REGION Network 4: Start Ejection
   #_w1 := #Current_machine_state = #st_finishing_molding_sub3;
   #Process_Simulation_Timers[3].TON(IN := #_w1, PT := #Process_Simulation_Timers[3].PT);
   IF #_w1 AND NOT #Process_Simulation_Timers[3].Q THEN
       "FC_change_machineState"(stop_request := #stop_request,
                               new_stateNo := #st_finishing_molding_sub3,
                               new_stateDescription := 'Mold is opening',
                               act_error_code := 0,
                               act_warning_code := 0,
                               act_stateNo => #Current_machine_state,
                               info_actStateNo => #StationInfo.StateNo,
                               info_actStateDescription => #StationInfo.StateDescription,
                               info_errorCode => #StationInfo.ErrorCode,
                               info_warningCode => #StationInfo.WarningCode);
   END_IF;
   IF #_w1 AND #Process_Simulation_Timers[3].Q THEN
       "FC_change_machineState"(stop_request := #stop_request,
                               new_stateNo := #st_cycle_completed,
                               new_stateDescription := 'Ejection is starting',
                               act_error_code := 0,
                               act_warning_code := 0,
                               act_stateNo => #Current_machine_state,
                               info_actStateNo => #StationInfo.StateNo,
                               info_actStateDescription => #StationInfo.StateDescription,
                               info_errorCode => #StationInfo.ErrorCode,
                               info_warningCode => #StationInfo.WarningCode);
   END_IF;
END_REGION
END_FUNCTION_BLOCK

// folder: Flow5_Checking_Target_Production

FUNCTION_BLOCK "FB_Checking_Target_Production"   // FB11, LAD
{ S7_Optimized_Access := 'TRUE' }
VERSION : 0.1
   VAR_INPUT
      target_quantity : UInt;
   END_VAR
   VAR_IN_OUT
      stop_request : Bool;
      Current_machine_state : UInt;
      Act_Production_Quantity : UInt;
      StationInfo : Struct
         StateNo : UInt;
         StateDescription : String;
         ErrorCode : UInt;
         ErrorDescription : String;
         WarningCode : UInt;
         WarninDescription : String;
         TotalProductionTime : Time;
         ProducedCount : UInt;
      END_STRUCT;
   END_VAR
   VAR
      temp_state : UInt;
      Timeout : Array[0..5] of IEC_TIMER;
      Process_Simulation_Timers : Array[0..20] of IEC_TIMER;
      aux_var1 : Bool;
   END_VAR
   VAR CONSTANT
      st_idle : UInt := 0;
      st_cycle_completed : UInt := 500;
      st_cycle_completed_sub1 : UInt := 501;
      st_cycle_completed_sub2 : UInt := 502;
      st_cycle_completed_sub3 : UInt := 503;
      st_cycle_completed_sub4 : UInt := 504;
      st_cycle_completed_sub5 : UInt := 505;
      st_cycle_completed_sub6 : UInt := 506;
      st_cycle_completed_sub7 : UInt := 507;
      st_cycle_completed_sub8 : UInt := 508;
      st_cycle_completed_sub9 : UInt := 509;
      st_checking_order_target : UInt := 600;
      st_checking_initial_safety : UInt := 200;
      st_order_finishing : UInt := 700;
   END_VAR
   VAR_TEMP   // added for the SCL form of the ladder/FBD networks
      _w1 : Bool;
   END_VAR
   // Process_Simulation_Timers[0].PT := T#3S;
   // Process_Simulation_Timers[1].PT := T#4S;
   // Process_Simulation_Timers[2].PT := T#10S;
   // Process_Simulation_Timers[3].PT := T#3S;
BEGIN

REGION Network 1
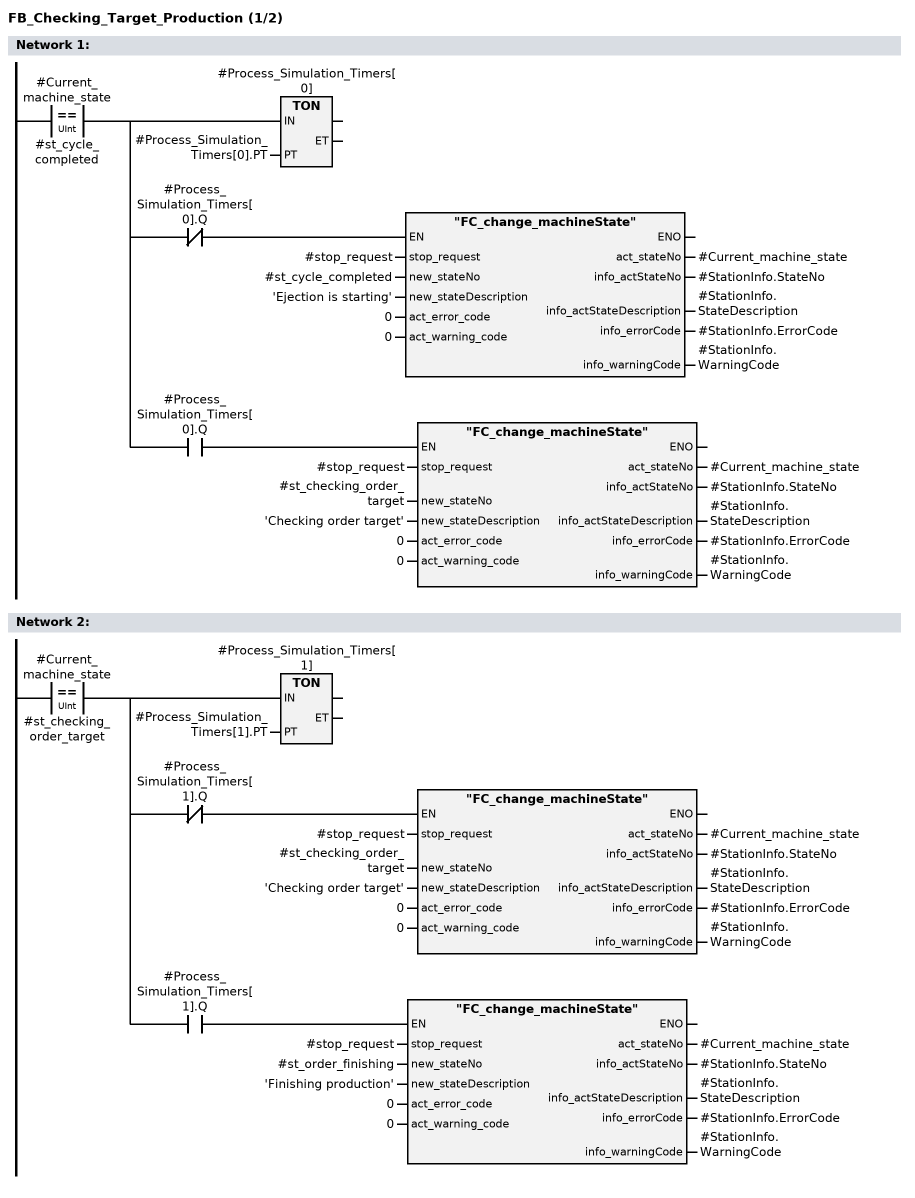
   #_w1 := #Current_machine_state = #st_cycle_completed;
   #Process_Simulation_Timers[0].TON(IN := #_w1, PT := #Process_Simulation_Timers[0].PT);
   IF #_w1 AND NOT #Process_Simulation_Timers[0].Q THEN
       "FC_change_machineState"(stop_request := #stop_request,
                               new_stateNo := #st_cycle_completed,
                               new_stateDescription := 'Ejection is starting',
                               act_error_code := 0,
                               act_warning_code := 0,
                               act_stateNo => #Current_machine_state,
                               info_actStateNo => #StationInfo.StateNo,
                               info_actStateDescription => #StationInfo.StateDescription,
                               info_errorCode => #StationInfo.ErrorCode,
                               info_warningCode => #StationInfo.WarningCode);
   END_IF;
   IF #_w1 AND #Process_Simulation_Timers[0].Q THEN
       "FC_change_machineState"(stop_request := #stop_request,
                               new_stateNo := #st_checking_order_target,
                               new_stateDescription := 'Checking order target',
                               act_error_code := 0,
                               act_warning_code := 0,
                               act_stateNo => #Current_machine_state,
                               info_actStateNo => #StationInfo.StateNo,
                               info_actStateDescription => #StationInfo.StateDescription,
                               info_errorCode => #StationInfo.ErrorCode,
                               info_warningCode => #StationInfo.WarningCode);
   END_IF;
END_REGION

REGION Network 2
   #_w1 := #Current_machine_state = #st_checking_order_target;
   #Process_Simulation_Timers[1].TON(IN := #_w1, PT := #Process_Simulation_Timers[1].PT);
   IF #_w1 AND NOT #Process_Simulation_Timers[1].Q THEN
       "FC_change_machineState"(stop_request := #stop_request,
                               new_stateNo := #st_checking_order_target,
                               new_stateDescription := 'Checking order target',
                               act_error_code := 0,
                               act_warning_code := 0,
                               act_stateNo => #Current_machine_state,
                               info_actStateNo => #StationInfo.StateNo,
                               info_actStateDescription => #StationInfo.StateDescription,
                               info_errorCode => #StationInfo.ErrorCode,
                               info_warningCode => #StationInfo.WarningCode);
   END_IF;
   IF #_w1 AND #Process_Simulation_Timers[1].Q THEN
       "FC_change_machineState"(stop_request := #stop_request,
                               new_stateNo := #st_order_finishing,
                               new_stateDescription := 'Finishing production',
                               act_error_code := 0,
                               act_warning_code := 0,
                               act_stateNo => #Current_machine_state,
                               info_actStateNo => #StationInfo.StateNo,
                               info_actStateDescription => #StationInfo.StateDescription,
                               info_errorCode => #StationInfo.ErrorCode,
                               info_warningCode => #StationInfo.WarningCode);
   END_IF;
END_REGION

REGION Network 3
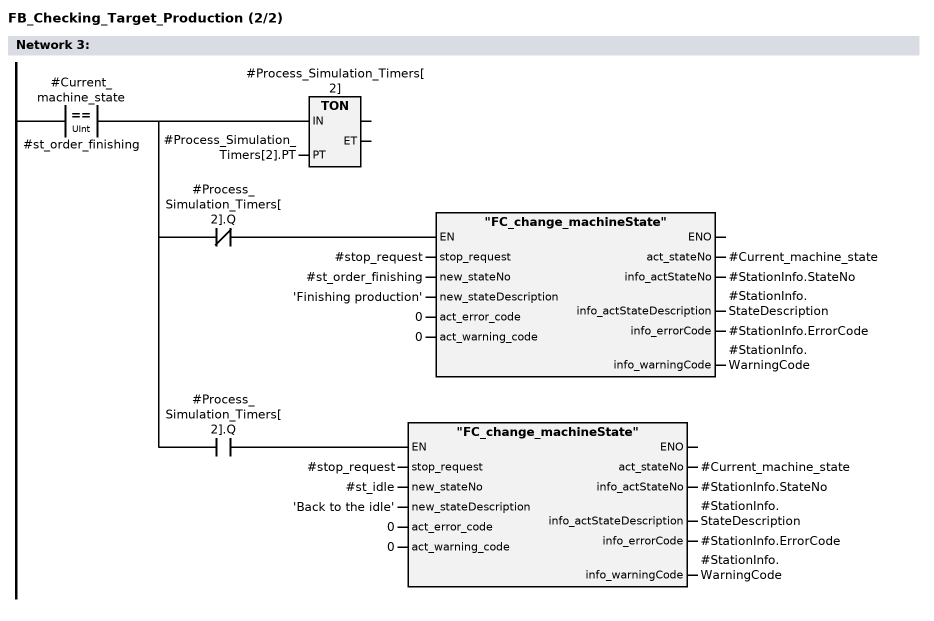
   #_w1 := #Current_machine_state = #st_order_finishing;
   #Process_Simulation_Timers[2].TON(IN := #_w1, PT := #Process_Simulation_Timers[2].PT);
   IF #_w1 AND NOT #Process_Simulation_Timers[2].Q THEN
       "FC_change_machineState"(stop_request := #stop_request,
                               new_stateNo := #st_order_finishing,
                               new_stateDescription := 'Finishing production',
                               act_error_code := 0,
                               act_warning_code := 0,
                               act_stateNo => #Current_machine_state,
                               info_actStateNo => #StationInfo.StateNo,
                               info_actStateDescription => #StationInfo.StateDescription,
                               info_errorCode => #StationInfo.ErrorCode,
                               info_warningCode => #StationInfo.WarningCode);
   END_IF;
   IF #_w1 AND #Process_Simulation_Timers[2].Q THEN
       "FC_change_machineState"(stop_request := #stop_request,
                               new_stateNo := #st_idle,
                               new_stateDescription := 'Back to the idle',
                               act_error_code := 0,
                               act_warning_code := 0,
                               act_stateNo => #Current_machine_state,
                               info_actStateNo => #StationInfo.StateNo,
                               info_actStateDescription => #StationInfo.StateDescription,
                               info_errorCode => #StationInfo.ErrorCode,
                               info_warningCode => #StationInfo.WarningCode);
   END_IF;
END_REGION
END_FUNCTION_BLOCK

// folder: Functions

FUNCTION "FC_get_time_data" : Void   // FC1, LAD
{ S7_Optimized_Access := 'TRUE' }
VERSION : 0.1
   VAR_OUTPUT
      actYear : UInt;
      actMonth : UInt;
      actDay : UInt;
      timeStamp : UDInt;
      errorGettingTime : Int;
   END_VAR
   VAR_TEMP
      timeData : DTL;
      gettingTimeState : Int;
   END_VAR
BEGIN

REGION Network 1
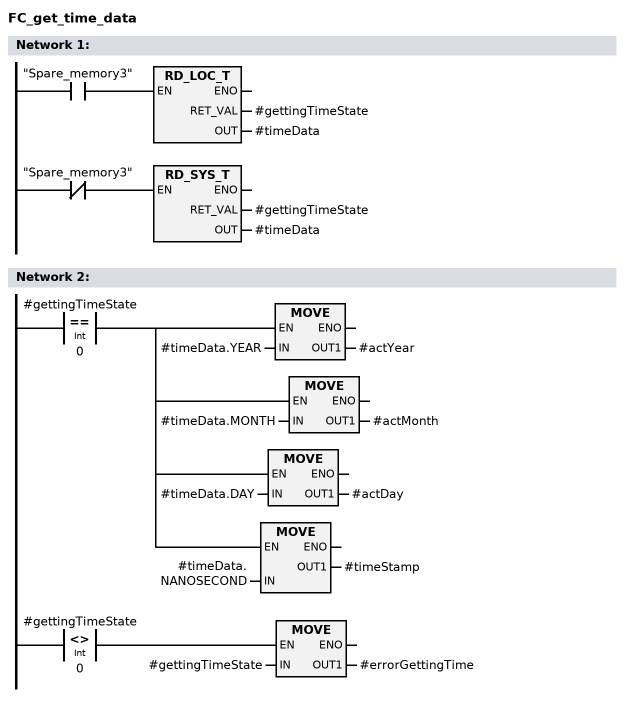
   IF "Spare_memory3" THEN #gettingTimeState := RD_LOC_T(OUT => #timeData); END_IF;
   IF NOT "Spare_memory3" THEN #gettingTimeState := RD_SYS_T(OUT => #timeData); END_IF;
END_REGION

REGION Network 2
   RUNG wire#powerrail
      { S7_Templates := "SrcType := Int" } EQ_Contact(in1 := #gettingTimeState, in2 := 0)
      wire#w1
      Move(in := #timeData.YEAR, out1 => #actYear)
   END_RUNG
   RUNG wire#w1
      Move(in := #timeData.MONTH, out1 => #actMonth)
   END_RUNG
   RUNG wire#w1
      Move(in := #timeData.DAY, out1 => #actDay)
   END_RUNG
   RUNG wire#w1
      Move(in := #timeData.NANOSECOND, out1 => #timeStamp)
   END_RUNG
   RUNG wire#powerrail
      { S7_Templates := "SrcType := Int" } NE_Contact(in1 := #gettingTimeState, in2 := 0)
      Move(in := #gettingTimeState, out1 => #errorGettingTime)
   END_RUNG
   // the same network as SCL:
   IF #gettingTimeState = 0 THEN
       #actYear := #timeData.YEAR;
       #actMonth := #timeData.MONTH;
       #actDay := #timeData.DAY;
       #timeStamp := #timeData.NANOSECOND;
   END_IF;
   IF #gettingTimeState <> 0 THEN #errorGettingTime := #gettingTimeState; END_IF;
END_REGION
END_FUNCTION

FUNCTION "FC_change_machineState" : Void   // FC2, LAD
{ S7_Optimized_Access := 'TRUE' }
VERSION : 0.1
   VAR_INPUT
      stop_request : Bool;
      new_stateNo : UInt;
      new_stateDescription : String;
      act_error_code : UInt;
      act_warning_code : UInt;
   END_VAR
   VAR_OUTPUT
      act_stateNo : UInt;
      info_actStateNo : UInt;
      info_actStateDescription : String;
      info_errorCode : UInt;
      info_warningCode : UInt;
   END_VAR
   VAR CONSTANT
      st_idle : UInt := 0;
   END_VAR
BEGIN

REGION Network 1: No Stop Request Received
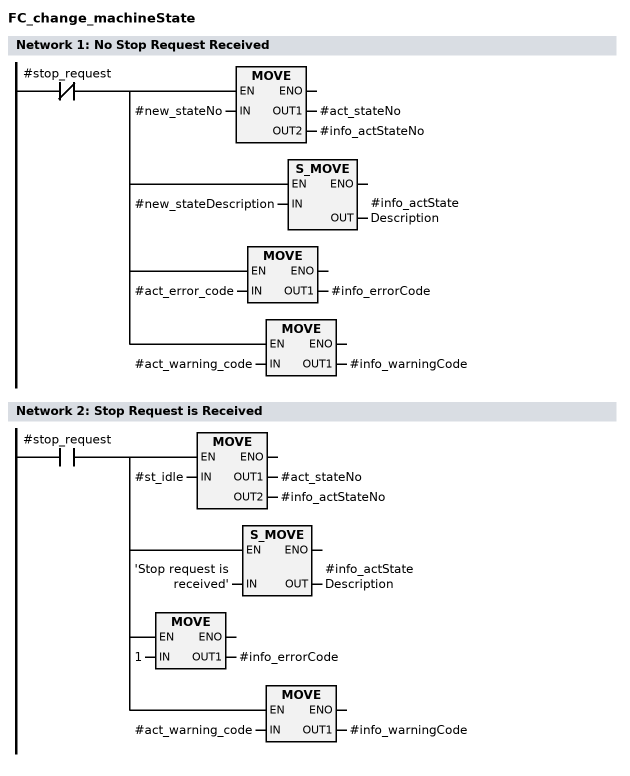
   RUNG wire#powerrail
      I_Contact( #stop_request )
      wire#w1
      Move(in := #new_stateNo, out1 => #act_stateNo, out2 => #info_actStateNo)
   END_RUNG
   RUNG wire#w1
      S_Move(in := #new_stateDescription, out => #info_actStateDescription)
   END_RUNG
   RUNG wire#w1
      Move(in := #act_error_code, out1 => #info_errorCode)
   END_RUNG
   RUNG wire#w1
      Move(in := #act_warning_code, out1 => #info_warningCode)
   END_RUNG
   // the same network as SCL:
   IF NOT #stop_request THEN
       #act_stateNo := #new_stateNo;
       #info_actStateNo := #new_stateNo;
       #info_actStateDescription := #new_stateDescription;
       #info_errorCode := #act_error_code;
       #info_warningCode := #act_warning_code;
   END_IF;
END_REGION

REGION Network 2: Stop Request is Received
   RUNG wire#powerrail
      Contact( #stop_request )
      wire#w1
      Move(in := #st_idle, out1 => #act_stateNo, out2 => #info_actStateNo)
   END_RUNG
   RUNG wire#w1
      S_Move(in := 'Stop request is received', out => #info_actStateDescription)
   END_RUNG
   RUNG wire#w1
      Move(in := 1, out1 => #info_errorCode)
   END_RUNG
   RUNG wire#w1
      Move(in := #act_warning_code, out1 => #info_warningCode)
   END_RUNG
   // the same network as SCL:
   IF #stop_request THEN
       #act_stateNo := #st_idle;
       #info_actStateNo := #st_idle;
       #info_actStateDescription := 'Stop request is received';
       #info_errorCode := 1;
       #info_warningCode := #act_warning_code;
   END_IF;
END_REGION
END_FUNCTION

// folder: Machine_transition

FUNCTION_BLOCK "FB_SubTransition"   // FB3, LAD
{ S7_Optimized_Access := 'TRUE' }
VERSION : 0.1
   VAR_INPUT
      new_state : UInt;
   END_VAR
   VAR_OUTPUT
      new_machine_state : UInt;
      previous_state_done : Bool;
   END_VAR
   VAR_IN_OUT
      stop_request : Bool;
   END_VAR
   VAR CONSTANT
      st_idle : UInt := 0;
   END_VAR
BEGIN

REGION Network 1: No Stop Request
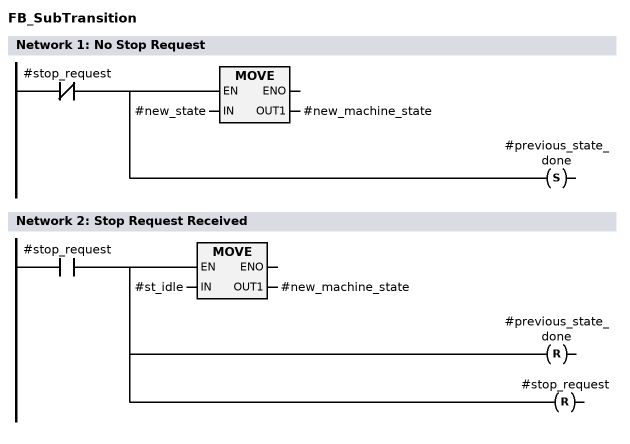
   RUNG wire#powerrail
      I_Contact( #stop_request )
      wire#w1
      Move(in := #new_state, out1 => #new_machine_state)
   END_RUNG
   RUNG wire#w1
      S_Coil( #previous_state_done )
   END_RUNG
   // the same network as SCL:
   IF NOT #stop_request THEN
       #new_machine_state := #new_state;
       #previous_state_done := TRUE;
   END_IF;
END_REGION

REGION Network 2: Stop Request Received
   RUNG wire#powerrail
      Contact( #stop_request )
      wire#w1
      Move(in := #st_idle, out1 => #new_machine_state)
   END_RUNG
   RUNG wire#w1
      R_Coil( #previous_state_done )
   END_RUNG
   RUNG wire#w1
      R_Coil( #stop_request )
   END_RUNG
   // the same network as SCL:
   IF #stop_request THEN
       #new_machine_state := #st_idle;
       #previous_state_done := FALSE;
       #stop_request := FALSE;
   END_IF;
END_REGION
END_FUNCTION_BLOCK

FUNCTION_BLOCK "FB_control_state_transition"   // FB6, LAD
TITLE = This FB sets the machine status
{ S7_Optimized_Access := 'TRUE' }
VERSION : 0.1
   VAR_INPUT
      is_start_btn_activated : Bool;
      is_stop_btn_activated : Bool;
   END_VAR
   VAR_IN_OUT
      current_machine_state : UInt;
      is_previous_state_done : Bool;
   END_VAR
   VAR
      temp_state : UInt;
      initial_temp_state : UInt;
      stop_request : Bool;
   END_VAR
   VAR CONSTANT
      st_idle : UInt := 0;
      st_checking_order : UInt := 10;
      st_checking_initial_safety : UInt := 20;
      st_checking_material_level : UInt := 30;
      st_running_molding : UInt := 40;
      st_finishing_molding : UInt := 50;
      st_cycle_completed : UInt := 60;
      st_checking_order_target : UInt := 70;
      st_order_finishing : UInt := 80;
      st_fault : UInt := 300;
   END_VAR
   VAR_TEMP   // added for the SCL form of the ladder/FBD networks
      _w1 : Bool;
   END_VAR
BEGIN

REGION Network 1: Control Stop Request
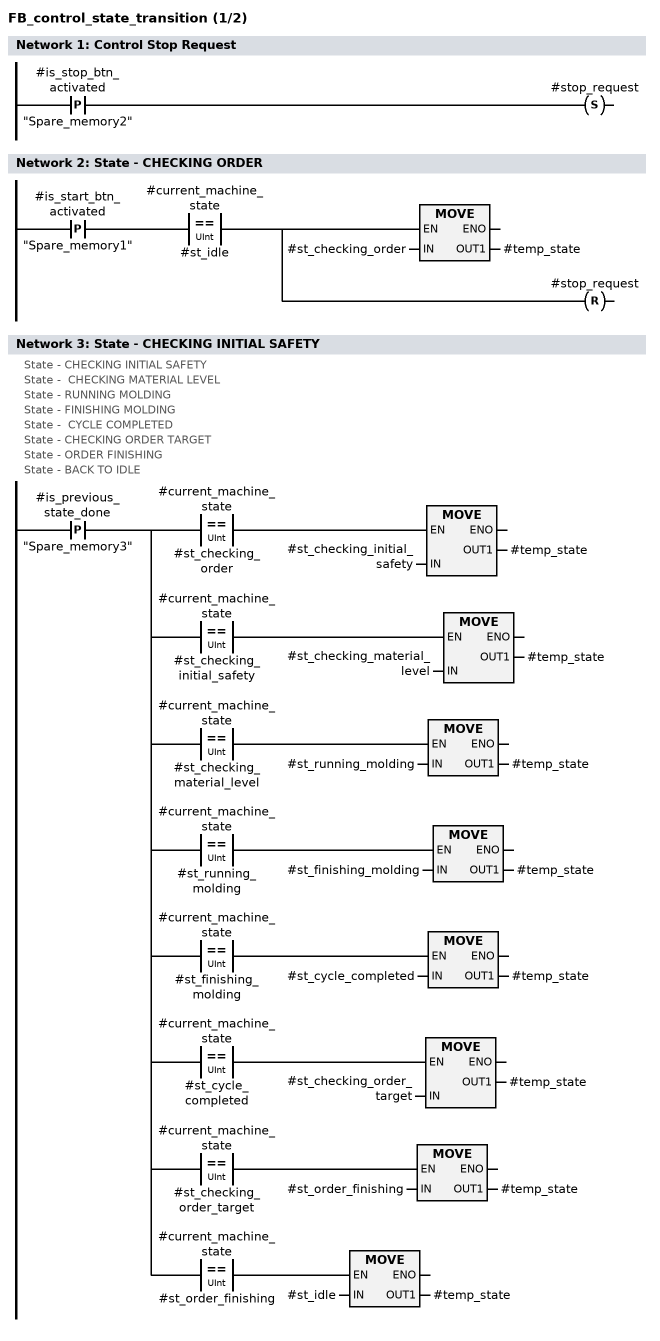
   RUNG wire#powerrail
      P_Contact(operand := #is_stop_btn_activated, bit := "Spare_memory2")
      S_Coil( #stop_request )
   END_RUNG
   // the same network as SCL:
   #_w1 := #is_stop_btn_activated AND NOT "Spare_memory2";   // rising edge of #is_stop_btn_activated
   "Spare_memory2" := #is_stop_btn_activated;
   IF #_w1 THEN #stop_request := TRUE; END_IF;
END_REGION

REGION Network 2: State - CHECKING ORDER
   RUNG wire#powerrail
      P_Contact(operand := #is_start_btn_activated, bit := "Spare_memory1")
      { S7_Templates := "SrcType := UInt" } EQ_Contact(in1 := #current_machine_state, in2 := #st_idle)
      wire#w1
      Move(in := #st_checking_order, out1 => #temp_state)
   END_RUNG
   RUNG wire#w1
      R_Coil( #stop_request )
   END_RUNG
   // the same network as SCL:
   #_w1 := #is_start_btn_activated AND NOT "Spare_memory1";   // rising edge of #is_start_btn_activated
   "Spare_memory1" := #is_start_btn_activated;
   IF #_w1 AND (#current_machine_state = #st_idle) THEN
       #temp_state := #st_checking_order;
       #stop_request := FALSE;
   END_IF;
END_REGION

REGION Network 3: State - CHECKING INITIAL SAFETY
   // State - CHECKING INITIAL SAFETY
   // State -  CHECKING MATERIAL LEVEL
   // State - RUNNING MOLDING
   // State - FINISHING MOLDING
   // State -  CYCLE COMPLETED
   // State - CHECKING ORDER TARGET
   // State - ORDER FINISHING 
   // State - BACK TO IDLE
   RUNG wire#powerrail
      P_Contact(operand := #is_previous_state_done, bit := "Spare_memory3")
      wire#w1
      { S7_Templates := "SrcType := UInt" } EQ_Contact(in1 := #current_machine_state, in2 := #st_checking_order)
      Move(in := #st_checking_initial_safety, out1 => #temp_state)
   END_RUNG
   RUNG wire#w1
      { S7_Templates := "SrcType := UInt" } EQ_Contact(in1 := #current_machine_state, in2 := #st_checking_initial_safety)
      Move(in := #st_checking_material_level, out1 => #temp_state)
   END_RUNG
   RUNG wire#w1
      { S7_Templates := "SrcType := UInt" } EQ_Contact(in1 := #current_machine_state, in2 := #st_checking_material_level)
      Move(in := #st_running_molding, out1 => #temp_state)
   END_RUNG
   RUNG wire#w1
      { S7_Templates := "SrcType := UInt" } EQ_Contact(in1 := #current_machine_state, in2 := #st_running_molding)
      Move(in := #st_finishing_molding, out1 => #temp_state)
   END_RUNG
   RUNG wire#w1
      { S7_Templates := "SrcType := UInt" } EQ_Contact(in1 := #current_machine_state, in2 := #st_finishing_molding)
      Move(in := #st_cycle_completed, out1 => #temp_state)
   END_RUNG
   RUNG wire#w1
      { S7_Templates := "SrcType := UInt" } EQ_Contact(in1 := #current_machine_state, in2 := #st_cycle_completed)
      Move(in := #st_checking_order_target, out1 => #temp_state)
   END_RUNG
   RUNG wire#w1
      { S7_Templates := "SrcType := UInt" } EQ_Contact(in1 := #current_machine_state, in2 := #st_checking_order_target)
      Move(in := #st_order_finishing, out1 => #temp_state)
   END_RUNG
   RUNG wire#w1
      { S7_Templates := "SrcType := UInt" } EQ_Contact(in1 := #current_machine_state, in2 := #st_order_finishing)
      Move(in := #st_idle, out1 => #temp_state)
   END_RUNG
   // the same network as SCL:
   #_w1 := #is_previous_state_done AND NOT "Spare_memory3";   // rising edge of #is_previous_state_done
   "Spare_memory3" := #is_previous_state_done;
   IF #_w1 AND (#current_machine_state = #st_checking_order) THEN
       #temp_state := #st_checking_initial_safety;
   END_IF;
   IF #_w1 AND (#current_machine_state = #st_checking_initial_safety) THEN
       #temp_state := #st_checking_material_level;
   END_IF;
   IF #_w1 AND (#current_machine_state = #st_checking_material_level) THEN
       #temp_state := #st_running_molding;
   END_IF;
   IF #_w1 AND (#current_machine_state = #st_running_molding) THEN
       #temp_state := #st_finishing_molding;
   END_IF;
   IF #_w1 AND (#current_machine_state = #st_finishing_molding) THEN
       #temp_state := #st_cycle_completed;
   END_IF;
   IF #_w1 AND (#current_machine_state = #st_cycle_completed) THEN
       #temp_state := #st_checking_order_target;
   END_IF;
   IF #_w1 AND (#current_machine_state = #st_checking_order_target) THEN
       #temp_state := #st_order_finishing;
   END_IF;
   IF #_w1 AND (#current_machine_state = #st_order_finishing) THEN #temp_state := #st_idle; END_IF;
END_REGION

REGION Network 4: Set the current machine state to new state value
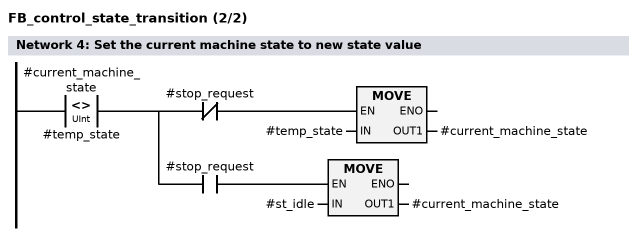
   RUNG wire#powerrail
      { S7_Templates := "SrcType := UInt" } NE_Contact(in1 := #current_machine_state, in2 := #temp_state)
      wire#w1
      I_Contact( #stop_request )
      Move(in := #temp_state, out1 => #current_machine_state)
   END_RUNG
   RUNG wire#w1
      Contact( #stop_request )
      Move(in := #st_idle, out1 => #current_machine_state)
   END_RUNG
   // the same network as SCL:
   #_w1 := #current_machine_state <> #temp_state;
   IF #_w1 AND NOT #stop_request THEN #current_machine_state := #temp_state; END_IF;
   IF #_w1 AND #stop_request THEN #current_machine_state := #st_idle; END_IF;
END_REGION
END_FUNCTION_BLOCK

// folder: Manage_outputs

FUNCTION_BLOCK "FB_manage_outputs"   // FB8, LAD
{ S7_Optimized_Access := 'TRUE' }
VERSION : 0.1
BEGIN

REGION Network 1: Feeder_Start
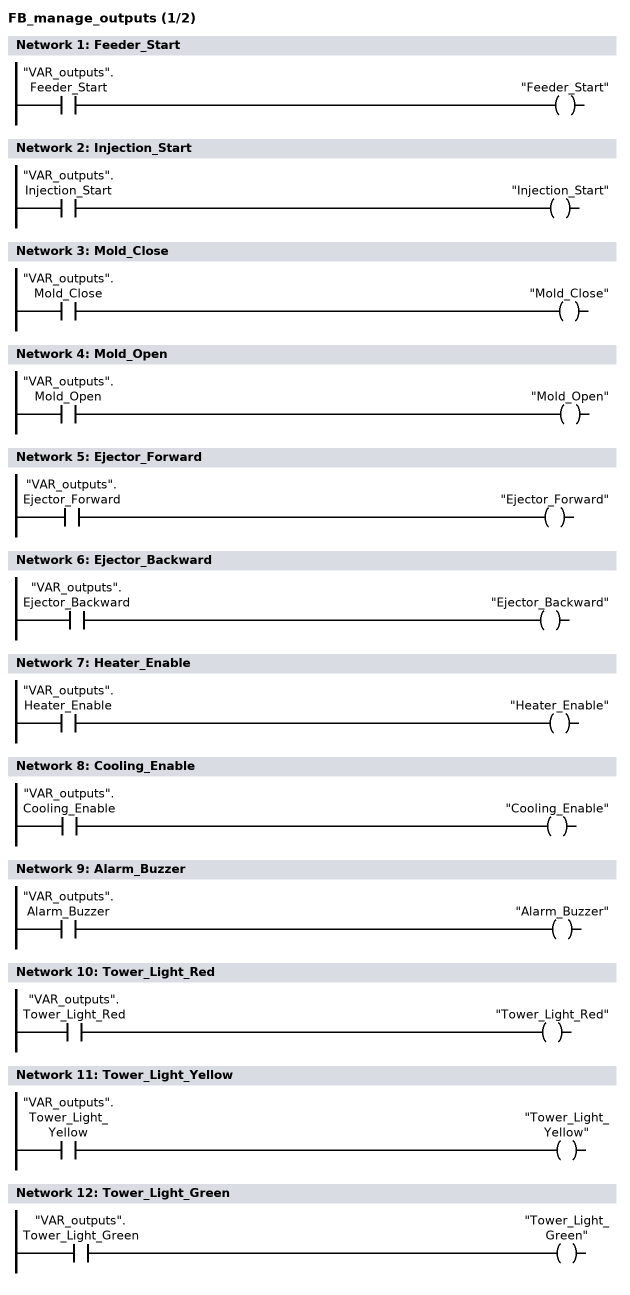
   RUNG wire#powerrail
      Contact( "VAR_outputs".Feeder_Start )
      Coil( "Feeder_Start" )
   END_RUNG
   // the same network as SCL:
   "Feeder_Start" := "VAR_outputs".Feeder_Start;
END_REGION

REGION Network 2: Injection_Start
   RUNG wire#powerrail
      Contact( "VAR_outputs".Injection_Start )
      Coil( "Injection_Start" )
   END_RUNG
   // the same network as SCL:
   "Injection_Start" := "VAR_outputs".Injection_Start;
END_REGION

REGION Network 3: Mold_Close
   RUNG wire#powerrail
      Contact( "VAR_outputs".Mold_Close )
      Coil( "Mold_Close" )
   END_RUNG
   // the same network as SCL:
   "Mold_Close" := "VAR_outputs".Mold_Close;
END_REGION

REGION Network 4: Mold_Open
   RUNG wire#powerrail
      Contact( "VAR_outputs".Mold_Open )
      Coil( "Mold_Open" )
   END_RUNG
   // the same network as SCL:
   "Mold_Open" := "VAR_outputs".Mold_Open;
END_REGION

REGION Network 5: Ejector_Forward
   RUNG wire#powerrail
      Contact( "VAR_outputs".Ejector_Forward )
      Coil( "Ejector_Forward" )
   END_RUNG
   // the same network as SCL:
   "Ejector_Forward" := "VAR_outputs".Ejector_Forward;
END_REGION

REGION Network 6: Ejector_Backward
   RUNG wire#powerrail
      Contact( "VAR_outputs".Ejector_Backward )
      Coil( "Ejector_Backward" )
   END_RUNG
   // the same network as SCL:
   "Ejector_Backward" := "VAR_outputs".Ejector_Backward;
END_REGION

REGION Network 7: Heater_Enable
   RUNG wire#powerrail
      Contact( "VAR_outputs".Heater_Enable )
      Coil( "Heater_Enable" )
   END_RUNG
   // the same network as SCL:
   "Heater_Enable" := "VAR_outputs".Heater_Enable;
END_REGION

REGION Network 8: Cooling_Enable
   RUNG wire#powerrail
      Contact( "VAR_outputs".Cooling_Enable )
      Coil( "Cooling_Enable" )
   END_RUNG
   // the same network as SCL:
   "Cooling_Enable" := "VAR_outputs".Cooling_Enable;
END_REGION

REGION Network 9: Alarm_Buzzer
   RUNG wire#powerrail
      Contact( "VAR_outputs".Alarm_Buzzer )
      Coil( "Alarm_Buzzer" )
   END_RUNG
   // the same network as SCL:
   "Alarm_Buzzer" := "VAR_outputs".Alarm_Buzzer;
END_REGION

REGION Network 10: Tower_Light_Red
   RUNG wire#powerrail
      Contact( "VAR_outputs".Tower_Light_Red )
      Coil( "Tower_Light_Red" )
   END_RUNG
   // the same network as SCL:
   "Tower_Light_Red" := "VAR_outputs".Tower_Light_Red;
END_REGION

REGION Network 11: Tower_Light_Yellow
   RUNG wire#powerrail
      Contact( "VAR_outputs".Tower_Light_Yellow )
      Coil( "Tower_Light_Yellow" )
   END_RUNG
   // the same network as SCL:
   "Tower_Light_Yellow" := "VAR_outputs".Tower_Light_Yellow;
END_REGION

REGION Network 12: Tower_Light_Green
   RUNG wire#powerrail
      Contact( "VAR_outputs".Tower_Light_Green )
      Coil( "Tower_Light_Green" )
   END_RUNG
   // the same network as SCL:
   "Tower_Light_Green" := "VAR_outputs".Tower_Light_Green;
END_REGION

REGION Network 13: Goto_NextStationBuffer
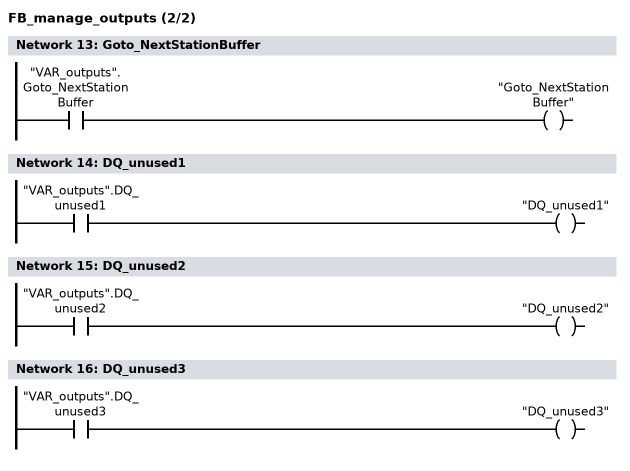
   RUNG wire#powerrail
      Contact( "VAR_outputs".Goto_NextStationBuffer )
      Coil( "Goto_NextStationBuffer" )
   END_RUNG
   // the same network as SCL:
   "Goto_NextStationBuffer" := "VAR_outputs".Goto_NextStationBuffer;
END_REGION

REGION Network 14: DQ_unused1
   RUNG wire#powerrail
      Contact( "VAR_outputs".DQ_unused1 )
      Coil( "DQ_unused1" )
   END_RUNG
   // the same network as SCL:
   "DQ_unused1" := "VAR_outputs".DQ_unused1;
END_REGION

REGION Network 15: DQ_unused2
   RUNG wire#powerrail
      Contact( "VAR_outputs".DQ_unused2 )
      Coil( "DQ_unused2" )
   END_RUNG
   // the same network as SCL:
   "DQ_unused2" := "VAR_outputs".DQ_unused2;
END_REGION

REGION Network 16: DQ_unused3
   RUNG wire#powerrail
      Contact( "VAR_outputs".DQ_unused3 )
      Coil( "DQ_unused3" )
   END_RUNG
   // the same network as SCL:
   "DQ_unused3" := "VAR_outputs".DQ_unused3;
END_REGION
END_FUNCTION_BLOCK

// folder: Simulation_data/Simulation_FB

FUNCTION_BLOCK "FB_simulate_analog_data"   // FB10, LAD
{ S7_Optimized_Access := 'TRUE' }
VERSION : 0.1
   VAR_INPUT
      Clock : Bool;
      Up : Bool;
      Down : Bool;
      TargetLevelLimit : Real;
      HighLevelLimit : Real;
      LowLevelLimit : Real;
      ResetVal : Bool;
   END_VAR
   VAR_IN_OUT
      actLevel : Real;
   END_VAR
   VAR
      value_int : Int;
      value_real : Real;
   END_VAR
   VAR_TEMP
      tag1 : Bool;
   END_VAR
   VAR CONSTANT
      incrementVal : Int := 5;
      decrementVal : Int := 150;
      normMin : Int := 0;
      normMax : Int := 27648;
   END_VAR
   VAR_TEMP   // added for the SCL form of the ladder/FBD networks
      _w1 : Bool;
   END_VAR
BEGIN

REGION Network 1: Simulate an analog input value
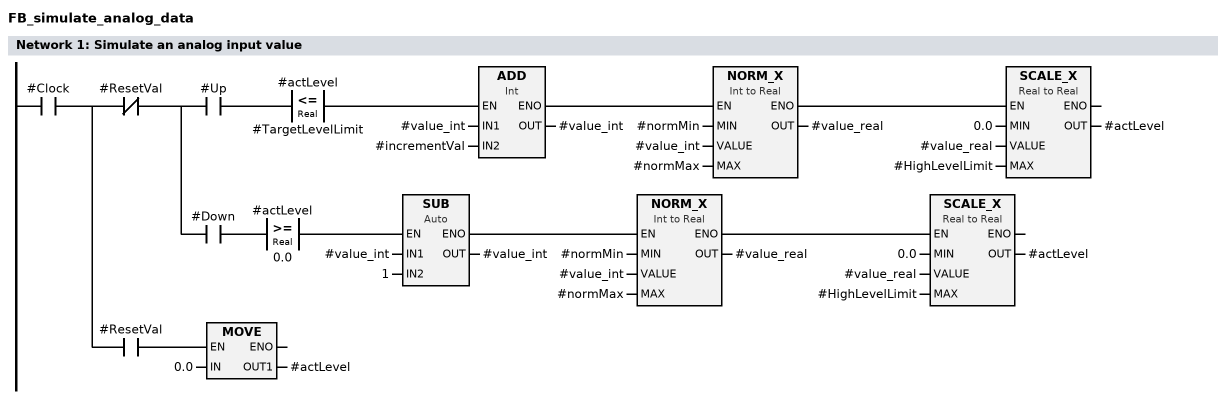
   RUNG wire#powerrail
      Contact( #Clock )
      wire#w1
      I_Contact( #ResetVal )
      wire#w2
      Contact( #Up )
      { S7_Templates := "SrcType := Real" } LE_Contact(in1 := #actLevel, in2 := #TargetLevelLimit)
      { S7_Templates := "SrcType := Int" } Add(in1 := #value_int, in2 := #incrementVal, out => #value_int)
      { S7_Templates := "[SrcType := Int, DestType := Real]" } Normalize(min := #normMin, value := #value_int, max := #normMax, out => #value_real)
      { S7_Templates := "[SrcType := Real, DestType := Real]" } Scale(min := 0.0, value := #value_real, max := #HighLevelLimit, out => #actLevel)
   END_RUNG
   RUNG wire#w2
      Contact( #Down )
      { S7_Templates := "SrcType := Real" } GE_Contact(in1 := #actLevel, in2 := 0.0)
      Sub(in1 := #value_int, in2 := 1, out => #value_int)
      { S7_Templates := "[SrcType := Int, DestType := Real]" } Normalize(min := #normMin, value := #value_int, max := #normMax, out => #value_real)
      { S7_Templates := "[SrcType := Real, DestType := Real]" } Scale(min := 0.0, value := #value_real, max := #HighLevelLimit, out => #actLevel)
   END_RUNG
   RUNG wire#w1
      Contact( #ResetVal )
      Move(in := 0.0, out1 => #actLevel)
   END_RUNG
   // the same network as SCL:
   #_w1 := #Clock AND NOT #ResetVal;
   IF #_w1 AND #Up AND (#actLevel <= #TargetLevelLimit) THEN
       #value_int := #value_int + #incrementVal;
       #value_real := NORM_X(MIN := #normMin, VALUE := #value_int, MAX := #normMax);
       #actLevel := SCALE_X(MIN := 0.0, VALUE := #value_real, MAX := #HighLevelLimit);
   END_IF;
   IF #_w1 AND #Down AND (#actLevel >= 0.0) THEN
       #value_int := #value_int - 1;
       #value_real := NORM_X(MIN := #normMin, VALUE := #value_int, MAX := #normMax);
       #actLevel := SCALE_X(MIN := 0.0, VALUE := #value_real, MAX := #HighLevelLimit);
   END_IF;
   IF #Clock AND #ResetVal THEN #actLevel := 0.0; END_IF;
END_REGION
END_FUNCTION_BLOCK

FUNCTION_BLOCK "FB_simulate_digital_input"   // FB16, LAD
{ S7_Optimized_Access := 'TRUE' }
VERSION : 0.1
   VAR_INPUT
      Open : Bool;
      Close : Bool;
   END_VAR
   VAR_IN_OUT
      Opened : Bool;
      Closed : Bool;
   END_VAR
   VAR
      Sim_timers : Array[0..2] of IEC_TIMER;
   END_VAR
   // Sim_timers[0].PT := T#5S;
   // Sim_timers[1].PT := T#5S;
BEGIN

REGION Network 1
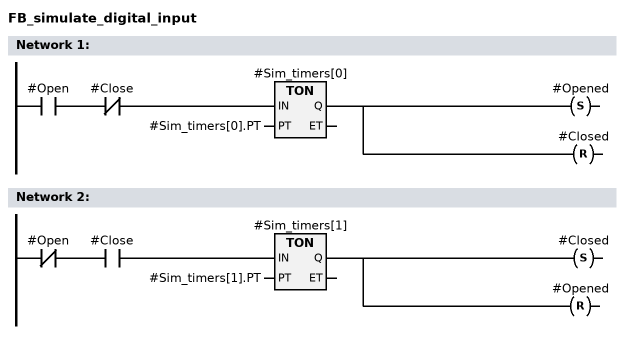
   #Sim_timers[0].TON(IN := #Open AND NOT #Close, PT := #Sim_timers[0].PT);
   IF #Sim_timers[0].Q THEN
       #Opened := TRUE;
       #Closed := FALSE;
   END_IF;
END_REGION

REGION Network 2
   #Sim_timers[1].TON(IN := NOT #Open AND #Close, PT := #Sim_timers[1].PT);
   IF #Sim_timers[1].Q THEN
       #Closed := TRUE;
       #Opened := FALSE;
   END_IF;
END_REGION
END_FUNCTION_BLOCK